FUNCTION_BLOCK SortingConveyor IMPLEMENTS I_Module
VAR
	_productDetected	:	I_Sensor;
	_conveyorFull	:	I_Sensor;
	_conveyorMotor	:	I_SingleDirectionMotor;
	_enabled	:	BOOL;
	_timeout: TOF;
END_VAR

_timeout(In := _enabled AND _productDetected.IsActive, PT := T#5S);

IF _enabled AND _timeout.Q AND NOT _conveyorFull.IsActive THEN
	_conveyorMotor.Start();
ELSE
	_conveyorMotor.Stop();
END_IF

METHOD Disable
VAR_INPUT
END_VAR
_enabled := false;
END_METHOD

METHOD Enable
VAR_INPUT
END_VAR
_enabled := true;
END_METHOD

METHOD FB_init : BOOL
VAR_INPUT
	bInitRetains : BOOL; // if TRUE, the retain variables are initialized (warm start / cold start)
	bInCopyCode : BOOL;  // if TRUE, the instance afterwards gets moved into the copy code (online change)
	ProductDetected	:	I_Sensor;
	ConveyorFull	:	I_Sensor;
	ConveyorMotor	:	I_SingleDirectionMotor;
END_VAR
// ATTENZIONE ALLO scope delle variabili !!
// usare THIS^ per dereferenziare le variabili locali 
// di questa istanza della classe SortingConveyor
THIS^._productDetected := ProductDetected;
THIS^._conveyorFull := ConveyorFull;
this^._conveyorMotor := ConveyorMotor;
END_METHOD

END_FUNCTION_BLOCK

(* stored: Version 1.1.0.1, ProductVersion 3.1.4024.11
   POU SortingConveyor: Id {6edeefe8-d3dc-4764-8536-d2ac7fc3a251}, SpecialFunc None
   Method Disable: Id {d21d1bad-9e97-409f-b2b3-4ec6e1e821c6}
   Method Enable: Id {f2c18022-b9d6-4908-833c-9365e754e1d7}
   Method FB_init: Id {265d8115-b619-48aa-a86a-c4d70b29ccbe} *)
